(* IEC 61131-3 sources: cds-text-sync-reference-project/project-view/PLC/PLC Logic/ST_Application/03_Object_POU_ST/02_FunctioanalBlock, 5 files *)

(* ---- ST_BLOCK_WITH_INTERFACE.st ---- *)
FUNCTION_BLOCK ST_BLOCK_WITH_INTERFACE
VAR_INPUT
	someBOOL : BOOL; //commentary
END_VAR
VAR_OUTPUT
END_VAR
VAR
END_VAR

(* ---- ST_FB.st ---- *)
FUNCTION_BLOCK ST_FB
VAR_INPUT
	xEnable : BOOL; // Enable counting
END_VAR
VAR_OUTPUT
	iCounter : INT; // Current counter value
	xLimitReached : BOOL; // Flag when limit is reached
END_VAR
VAR
	_iLimit : INT := 100; // Internal limit
END_VAR

// --- implementation ---

IF xEnable THEN
	IF iCounter < _iLimit THEN
		iCounter := iCounter + 1;
		xLimitReached := FALSE;
	ELSE
		xLimitReached := TRUE;
	END_IF
ELSE
	xLimitReached := FALSE;
END_IF

(* ---- ST_FB.ST_FB_Method.st ---- *)
METHOD ST_FB_Method : BOOL
VAR_INPUT
	iValueToAdd : INT;
END_VAR

// --- implementation ---

IF (iCounter + iValueToAdd) <= _iLimit THEN
	iCounter := iCounter + iValueToAdd;
	ST_FB_Method := TRUE;
ELSE
	ST_FB_Method := FALSE;
END_IF

(* ---- ST_FB.ST_FB_Property.Get.st ---- *)
VAR
END_VAR

// --- implementation ---

ST_FB_Property := _iLimit;

(* ---- ST_FB.ST_FB_Property.Set.st ---- *)
VAR
END_VAR

// --- implementation ---

_iLimit := ST_FB_Property;
